// Mitsubishi GX Works2 project: 세척,열풍건조, 동결건조_테스트   PLC: Q02U

PROGRAM INPUT
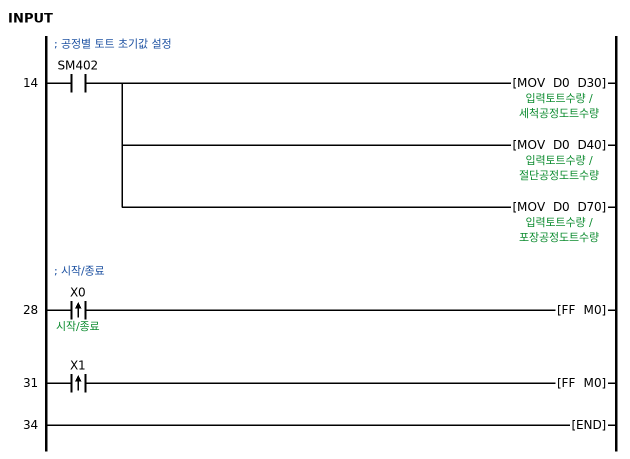
; 공정별 토트 초기값 설정
14    LD      SM402
      MOV     D0 D30  ; 입력토트수량 / 세척공정도트수량
      MOV     D0 D40  ; 절단공정도트수량
      MOV     D0 D70  ; 포장공정도트수량
; 시작/종료
28    LDP     X0  ; 시작/종료
      FF      M0
31    LDP     X1
      FF      M0
34    END
END_PROGRAM

PROGRAM 세척공정
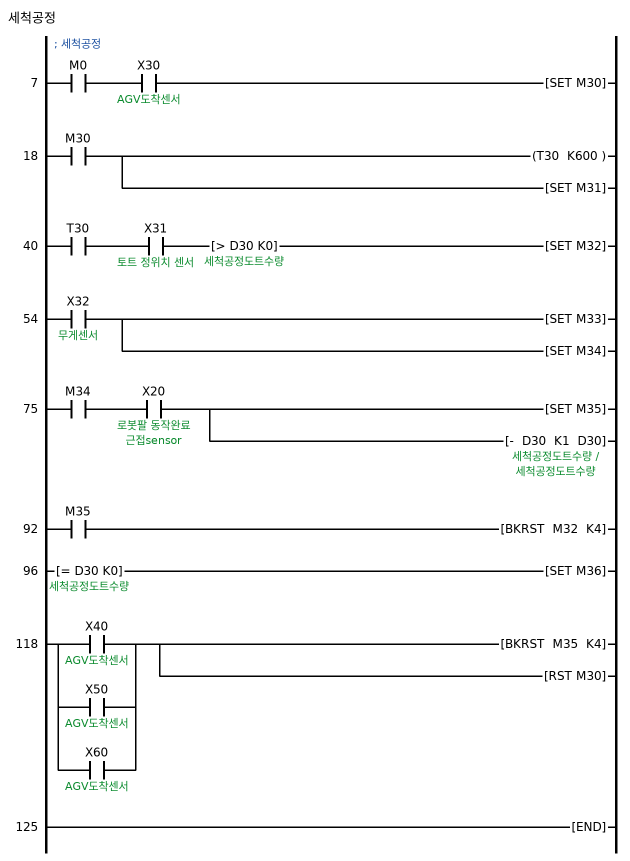
; 세척공정
7     LD      M0
      AND     X30  ; AGV도착센서
      SET     M30
        [note] 펌프모터 ON
18    LD      M30
      OUT     T30 K600
        [note] 펌핑모터 OFF
      SET     M31
        [note] SubCVY ON
40    LD      T30
      AND     X31  ; 토트 정위치 센서
      AND>    D30 K0  ; 세척공정도트수량
      SET     M32
        [note] MainCVY ON
54    LD      X32  ; 무게센서
      SET     M33
        [note] MAinCVY OFF
      SET     M34
        [note] 하역 로봇팔 ON
75    LD      M34
      AND     X20  ; 로봇팔 동작완료 근접sensor
      SET     M35
        [note] 하역 로봇팔 OFF
      -       D30 K1 D30
92    LD      M35
      BKRST   M32 K4
96    LD=     D30 K0  ; 세척공정도트수량
      SET     M36
        [note] AGV 다음 공정 이동, SubCVY OFF
118   LD      X40  ; AGV도착센서
      OR      X50  ; AGV도착센서
      OR      X60  ; AGV도착센서
      BKRST   M35 K4
      RST     M30
125   END
END_PROGRAM

PROGRAM 열풍건조
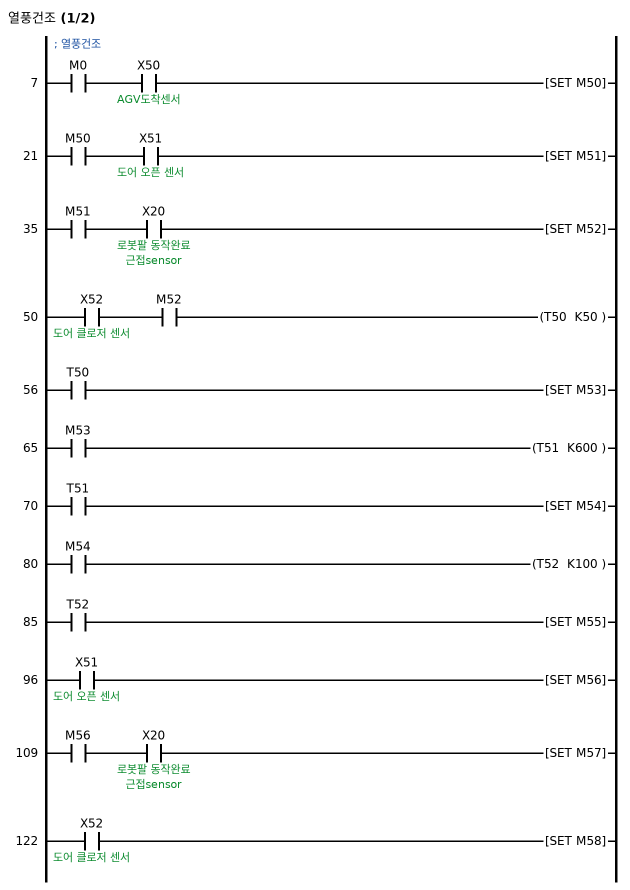
; 열풍건조
7     LD      M0
      AND     X50  ; AGV도착센서
      SET     M50
        [note] 도어 오픈모터(정)
21    LD      M50
      AND     X51  ; 도어 오픈 센서
      SET     M51
        [note] 상역 로봇 팔동작
35    LD      M51
      AND     X20  ; 로봇팔 동작완료 근접sensor
      SET     M52
        [note] 도어 클로즈모터(정)
50    LD      X52  ; 도어 클로저 센서
      AND     M52
      OUT     T50 K50
56    LD      T50
      SET     M53
        [note] 건조기 ON
65    LD      M53
      OUT     T51 K600
70    LD      T51
      SET     M54
        [note] 건조기 OFF
80    LD      M54
      OUT     T52 K100
85    LD      T52
      SET     M55
        [note] 도어 오픈CYL
96    LD      X51  ; 도어 오픈 센서
      SET     M56
        [note] 하역 로봇팔 동작
109   LD      M56
      AND     X20  ; 로봇팔 동작완료 근접sensor
      SET     M57
        [note] 도어 클로즈CYL
122   LD      X52  ; 도어 클로저 센서
      SET     M58
        [note] AGV 다음 공정 이동
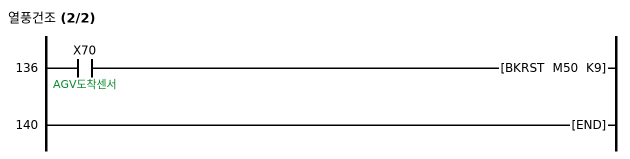
136   LD      X70  ; AGV도착센서
      BKRST   M50 K9
140   END
END_PROGRAM

PROGRAM OUTPUT
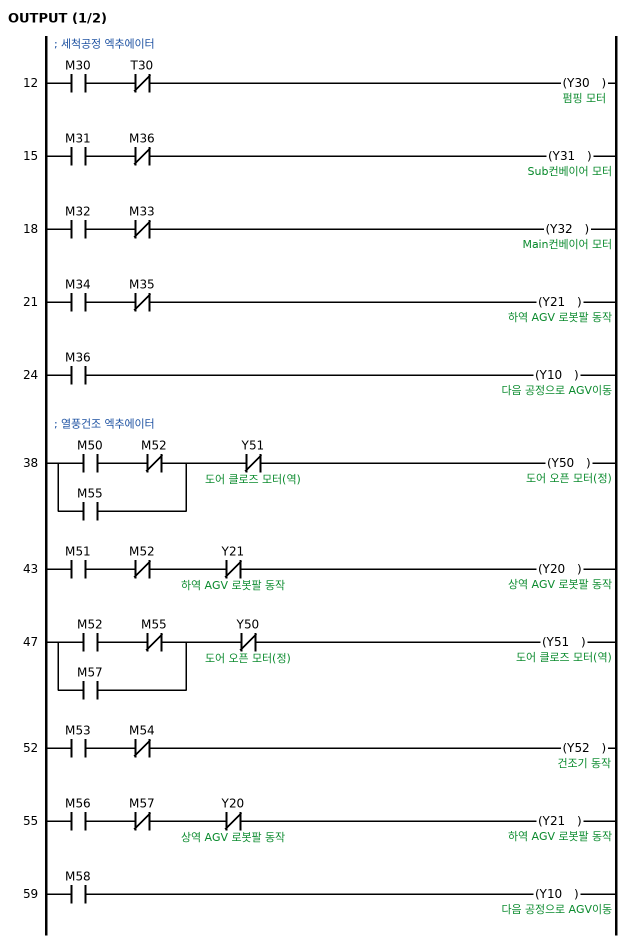
; 세척공정 엑추에이터
12    LD      M30
      ANI     T30
      OUT     Y30  ; 펌핑 모터
15    LD      M31
      ANI     M36
      OUT     Y31  ; Sub컨베이어 모터
18    LD      M32
      ANI     M33
      OUT     Y32  ; Main컨베이어 모터
21    LD      M34
      ANI     M35
      OUT     Y21  ; 하역 AGV 로봇팔 동작
24    LD      M36
      OUT     Y10  ; 다음 공정으로 AGV이동
; 열풍건조 엑추에이터
38    LD      M50
      ANI     M52
      OR      M55
      ANI     Y51  ; 도어 클로즈 모터(역)
      OUT     Y50  ; 도어 오픈 모터(정)
43    LD      M51
      ANI     M52
      ANI     Y21  ; 하역 AGV 로봇팔 동작
      OUT     Y20  ; 상역 AGV 로봇팔 동작
47    LD      M52
      ANI     M55
      OR      M57
      ANI     Y50  ; 도어 오픈 모터(정)
      OUT     Y51  ; 도어 클로즈 모터(역)
52    LD      M53
      ANI     M54
      OUT     Y52  ; 건조기 동작
55    LD      M56
      ANI     M57
      ANI     Y20  ; 상역 AGV 로봇팔 동작
      OUT     Y21  ; 하역 AGV 로봇팔 동작
59    LD      M58
      OUT     Y10  ; 다음 공정으로 AGV이동
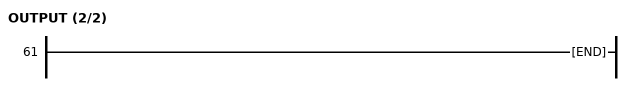
61    END
END_PROGRAM

PROGRAM 동결건조
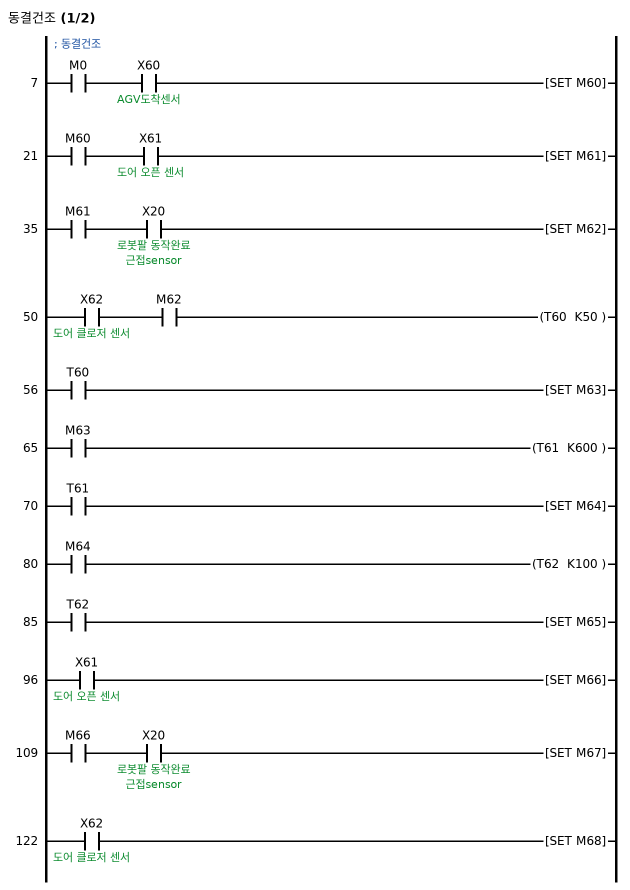
; 동결건조
7     LD      M0
      AND     X60  ; AGV도착센서
      SET     M60
        [note] 도어 오픈모터(정)
21    LD      M60
      AND     X61  ; 도어 오픈 센서
      SET     M61
        [note] 상역 로봇 팔동작
35    LD      M61
      AND     X20  ; 로봇팔 동작완료 근접sensor
      SET     M62
        [note] 도어 클로즈모터(정)
50    LD      X62  ; 도어 클로저 센서
      AND     M62
      OUT     T60 K50
56    LD      T60
      SET     M63
        [note] 건조기 ON
65    LD      M63
      OUT     T61 K600
70    LD      T61
      SET     M64
        [note] 건조기 OFF
80    LD      M64
      OUT     T62 K100
85    LD      T62
      SET     M65
        [note] 도어 오픈CYL
96    LD      X61  ; 도어 오픈 센서
      SET     M66
        [note] 하역 로봇팔 동작
109   LD      M66
      AND     X20  ; 로봇팔 동작완료 근접sensor
      SET     M67
        [note] 도어 클로즈CYL
122   LD      X62  ; 도어 클로저 센서
      SET     M68
        [note] AGV 다음 공정 이동
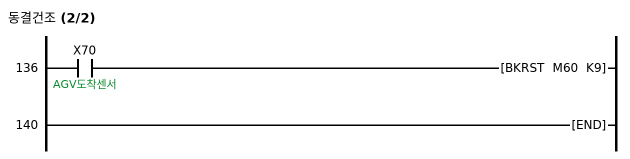
136   LD      X70  ; AGV도착센서
      BKRST   M60 K9
140   END
END_PROGRAM

PROGRAM 절단공정
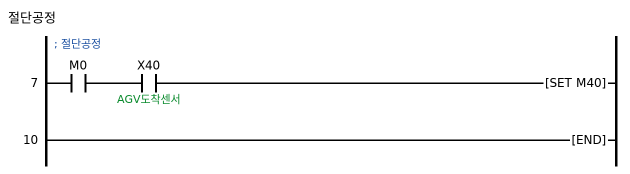
; 절단공정
7     LD      M0
      AND     X40  ; AGV도착센서
      SET     M40
10    END
END_PROGRAM

// device comments not shown above
X12  ; 토틀 감지 센서
Y60  ; 도어 오픈 모터(정)
Y61  ; 도어 클로즈 모터(역)
Y62  ; 건조기 동작
D50  ; 열풍건조공정도트수량
D60  ; 동결건조공정도트수량
